// TIA Portal V20 export
VAR_GLOBAL   // PLC tag table "ConvConstantB1"
END_VAR
VAR_GLOBAL CONSTANT   // user constants
   minB1 : Int := 2001;
   maxB1 : Int := 2002;
END_VAR
